{attribute 'strict'}
TYPE E_CR800StateSendPosition :
(
	CR800_SEND_POSITION_CONVERTING				:= 0,	(* DUMMY *)
	CR800_SEND_POSITION_SENDING					:= 10
); 
END_TYPE

(* stored: Version 1.1.0.1, ProductVersion 3.1.4024.9
   DUT E_CR800StateSendPosition: Id {0012320f-8cbb-4cd8-99ad-f6ddb8f13814} *)
